(* CODESYS project Ex_3.project

Project tree, tasks and I/O mapping:
  Device : CODESYS Control Win V3, 3S - Smart Software Solutions GmbH, version 3.5.20.50
    application Application
      libraries: Standard, 3.5.18.0 (System)
      task MainTask (cyclic, interval t#20ms, priority 1) calls PLC_PRG
      program PLC_PRG [ST]
*)

// Device/Application/PLC_PRG
PROGRAM PLC_PRG
VAR
	timer1:TON;
	start:BOOL;
	motor:BOOL;
	elapsedTime:TIME;
END_VAR

timer1(IN:=start, PT:=T#10S);
elapsedTime:=timer1.ET;
motor:=timer1.Q;
IF start=TRUE THEN
	timer1.IN:=TRUE;
ELSE
	timer1.IN:=FALSE;
END_IF

END_PROGRAM
